Staubli VAL3: COGNEX2.dtx

public bool bCalibrating
public bool bTaskDetOK
num hCamTable = 1
num nLatchedValue
public num nMaxNumOfObject = 10
public num nNumOfPart = -1
num nObjectID = -1
object oTempQueue
  [0]
    num nID
    trsf trTrsf
    num nLatchedValue
sio skVision
string sDetNum
string sTASK
string strError
trsf trObjectPos
